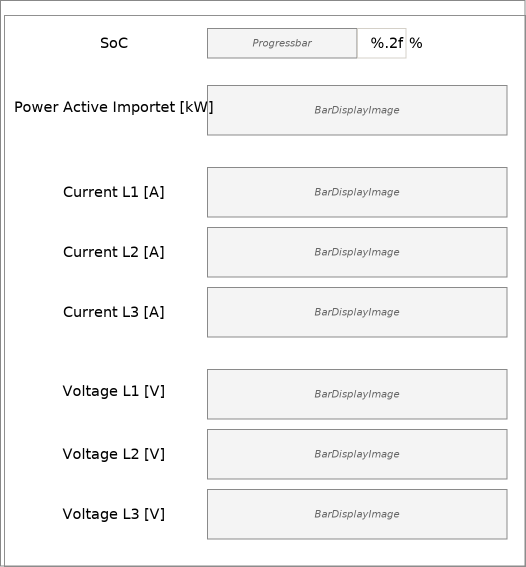
VISUALIZATION Measurand  // 526x567
VAR_IN_OUT
	fbMeasurand : FB_SampledValueMeasurands; 
END_VAR
    GroupBox (4,7 522x560)
        BarDisplayImage (203,160 300x50), value: fbMeasurand.fCurrentImportL1, style: BarDisplayImage-Gray, scale format: %.1f, scale 0..32
        Progressbar (203,21 150x30), variable: fbMeasurand.fStateOfCharge
        Textfield (353,21 49x30), "%.2f", text variable: fbMeasurand.fStateOfCharge
        Label (35,160 150x50), "Current L1 [A]"
        Label (35,220 150x50), "Current L2 [A]"
        Label (35,280 150x50), "Current L3 [A]"
        BarDisplayImage (203,362 300x50), value: fbMeasurand.fVoltageL1N, style: BarDisplayImage-Gray, scale format: %.1f, scale 0..250
        Label (35,362 150x44), "Voltage L1 [V]"
        Label (35,422 150x50), "Voltage L2 [V]"
        Label (35,482 150x50), "Voltage L3 [V]"
        Label (35,21 150x30), "SoC"
        BarDisplayImage (203,78 300x50), value: fbMeasurand.fPowerActiveImport, style: BarDisplayImage-Gray, scale format: %.1f, scale 0..22
        Label (35,85 150x30), "Power Active Importet [kW]"
        BarDisplayImage (203,220 300x50), value: fbMeasurand.fCurrentImportL2, style: BarDisplayImage-Gray, scale format: %.1f, scale 0..32
        BarDisplayImage (203,280 300x50), value: fbMeasurand.fCurrentImportL3, style: BarDisplayImage-Gray, scale format: %.1f, scale 0..32
        BarDisplayImage (203,422 300x50), value: fbMeasurand.fVoltageL2N, style: BarDisplayImage-Gray, scale format: %.1f, scale 0..250
        BarDisplayImage (203,482 300x50), value: fbMeasurand.fVoltageL3N, style: BarDisplayImage-Gray, scale format: %.1f, scale 0..250
        Label (402,21 47x30), "%"
END_VISUALIZATION

(* stored: Version 1.1.0.1
   Visu Measurand: Id {e320d245-9ff9-402c-95fc-05b7911573c5} *)
